Staubli VAL3: iIdent3.pgx

public program iIdent3(num& nNum[] (dimensions=1))
begin
  nNum=dioGet(iIdent3)
end
